// TIA Portal V15.1 export
// export: Created 2024-06-21T08:41:08.6869116Z, ExportSetting WithDefaults, DisplayName Totally Integrated Automation Portal, DisplayVersion V15.1 Update 5, DisplayName TIA Portal Openness, DisplayVersion V15.1 Update 5, DisplayName SINAMICS Startdrive Advanced, DisplayVersion V15.1, DisplayName G130, G150, S120, S150, SINAMICS MV, S210, DisplayVersion V15.1, DisplayName G110M, G120, G120C, G120D, G120P, DisplayVersion V15.1, DisplayName STEP 7 Professional, DisplayVersion V15.1 Update 5, DisplayName STEP 7 Safety, DisplayVersion V15.1, DisplayName WinCC Professional, DisplayVersion V15.1 Update 5, DisplayName SIMATIC Visualization Architect, DisplayVersion V15.1
FUNCTION "LGBHoist5PosIAnim" : Void   // FC6622, FBD
TITLE = LIAnimDWord / LGBHoist5PosIAnim
{ S7_Optimized_Access := 'TRUE' }
AUTHOR : VCC
FAMILY : Anim
NAME : SIAnim
VERSION : 0.1
// =============================================================================
// Handles the conversion from bits to one Word for simple icon Animation. 
// =============================================================================
// stored: AutoNumber false, IsIECCheckEnabled false, SetENOAutomatically False, UDAEnableTagReadback false
   VAR_INPUT
      I_OnPos : Bool;   // Set position / Set Position / On Position
      I_Active : Bool;   // Active
      I_Visible : Bool;   // ObjectVisible
      I_OutOfUse : Bool;   // Object out of use
      I_IntlkPos1 : Bool;   // Interlock for Set direction / Interlock for Position 1
      I_IntlkPos2 : Bool;   // Interlock for Set direction / Interlock for Position 2
      I_IntlkPos3 : Bool;   // Interlock for Reset direction / Interlock for Position 3
      I_IntlkPos4 : Bool;   // Interlock for Reset direction / Interlock for Position 4
      I_IntlkPos5 : Bool;   // Interlock for Reset direction / Interlock for Position 5
      I_IntlkPosMaint : Bool;   // Interlock for Reset direction / Interlock for Position Maintenance
      I_IntlkJog : Bool;   // Interlock for Reset direction / Interlock for Jog mode
      I_IntlkReferencing : Bool;   // Interlock for Reset direction / Interlock for Referencing mode
      I_VisibleIntlkPos1 : Bool;   // Interlock alarm for Set direction / Interlock Alarm for Set direction / Visible Interlock Position 1
      I_VisibleIntlkPos2 : Bool;   // Interlock alarm for Set direction / Interlock Alarm for Set direction / Visible Interlock Position 2
      I_VisibleIntlkPos3 : Bool;   // Interlock alarm for Reset direction / Interlock Alarm for Reset direction / Visible Interlock Position 3
      I_VisibleIntlkPos4 : Bool;   // Interlock alarm for Reset direction / Interlock Alarm for Reset direction / Visible Interlock Position 4
      I_VisibleIntlkPos5 : Bool;   // Interlock alarm for Reset direction / Interlock Alarm for Reset direction / Visible Interlock Position 5
      I_VisibleIntlkPosMaint : Bool;   // Interlock alarm for Reset direction / Interlock Alarm for Reset direction / Visible Interlock Position Maint
      I_ManualMode : Bool;   // Manual mode / Manual Mode
      I_FncSelInHMI : Bool;   // Manual selection from HMI
      I_AlarmA : Bool;   // AlarmA
      I_AlarmB : Bool;   // AlarmB
      I_AlarmC : Bool;   // AlarmC
      I_AlarmD : Bool;   // AlarmD
      I_SafetyOk : Bool;   // Safety Ok / Safety OK
      I_MotionStopNOk : Bool;   // Safety Ok / Motion Stop OK
   END_VAR
   VAR_OUTPUT
      H_IAnim : DWord;   // Icon animation Word / Icon Animation
   END_VAR
BEGIN

REGION Network 1: Icon animation Word / **** 1 - Inputs **** Set position / **** 1 - Inputs **** On position
   // Set Position / On position
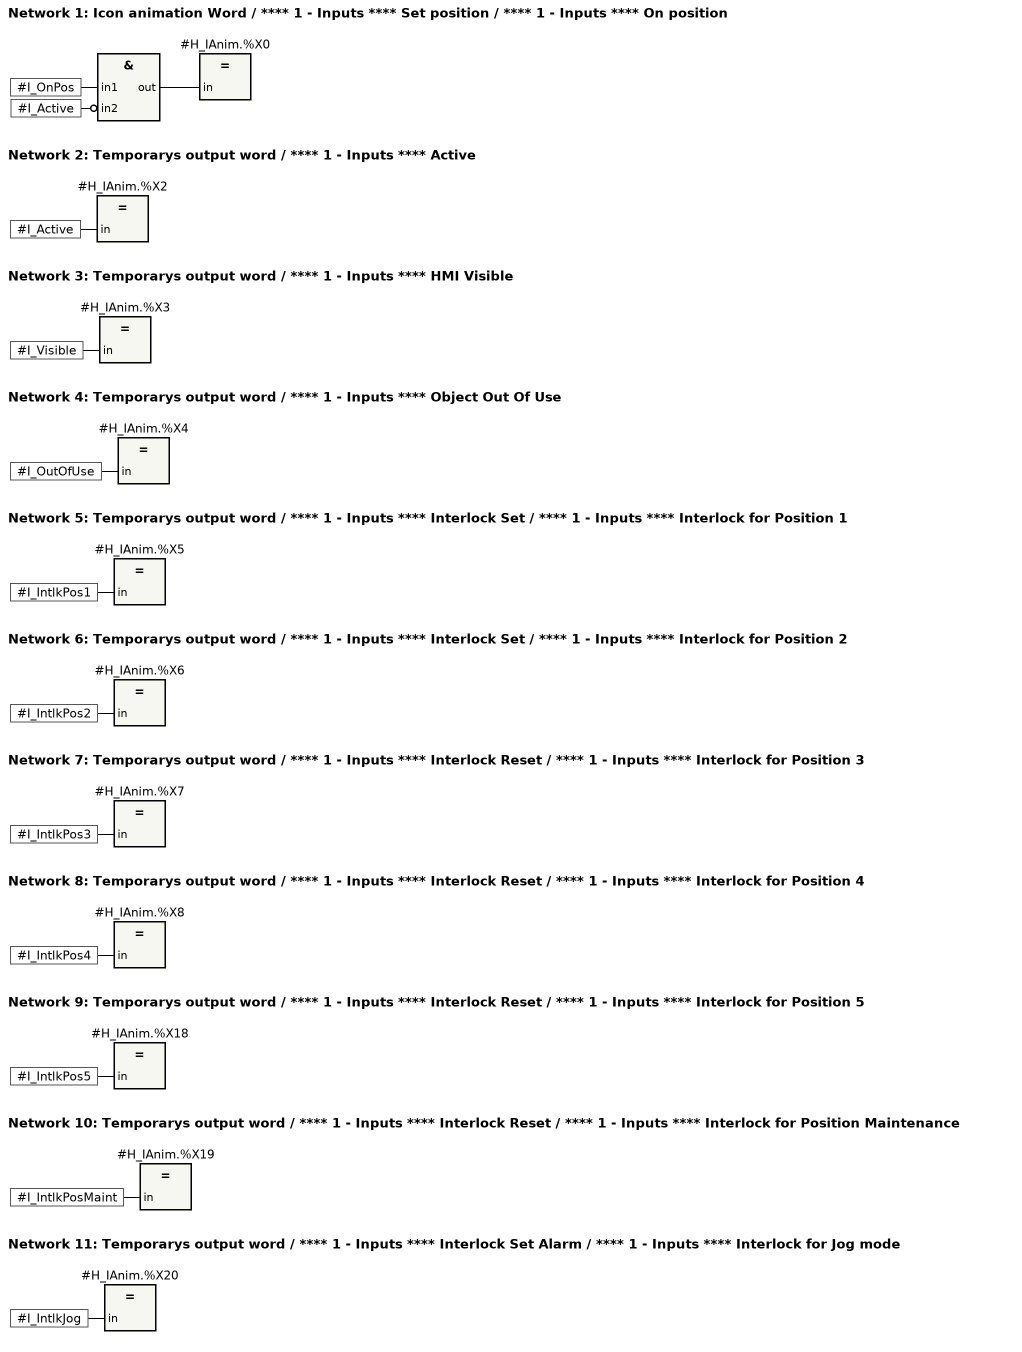
   #H_IAnim.%X0 := #I_OnPos AND NOT #I_Active;
END_REGION

REGION Network 2: Temporarys output word / **** 1 - Inputs **** Active
   // Active
   #H_IAnim.%X2 := #I_Active;
END_REGION

REGION Network 3: Temporarys output word / **** 1 - Inputs **** HMI Visible
   // HMI Visible
   #H_IAnim.%X3 := #I_Visible;
END_REGION

REGION Network 4: Temporarys output word / **** 1 - Inputs **** Object Out Of Use
   // Object out of use
   #H_IAnim.%X4 := #I_OutOfUse;
END_REGION

REGION Network 5: Temporarys output word / **** 1 - Inputs **** Interlock Set / **** 1 - Inputs **** Interlock for Position 1
   // Interlock Set / Interlock for Position 1
   #H_IAnim.%X5 := #I_IntlkPos1;
END_REGION

REGION Network 6: Temporarys output word / **** 1 - Inputs **** Interlock Set / **** 1 - Inputs **** Interlock for Position 2
   // Interlock Set / Interlock for Position 2
   #H_IAnim.%X6 := #I_IntlkPos2;
END_REGION

REGION Network 7: Temporarys output word / **** 1 - Inputs **** Interlock Reset / **** 1 - Inputs **** Interlock for Position 3
   // Interlock Reset / Interlock for Position 3
   #H_IAnim.%X7 := #I_IntlkPos3;
END_REGION

REGION Network 8: Temporarys output word / **** 1 - Inputs **** Interlock Reset / **** 1 - Inputs **** Interlock for Position 4
   // Interlock Reset / Interlock for Position 4
   #H_IAnim.%X8 := #I_IntlkPos4;
END_REGION

REGION Network 9: Temporarys output word / **** 1 - Inputs **** Interlock Reset / **** 1 - Inputs **** Interlock for Position 5
   // Interlock Reset / Interlock for Position 5
   #H_IAnim.%X18 := #I_IntlkPos5;
END_REGION

REGION Network 10: Temporarys output word / **** 1 - Inputs **** Interlock Reset / **** 1 - Inputs **** Interlock for Position Maintenance
   // Interlock Reset / Interlock for Position Maintenance
   #H_IAnim.%X19 := #I_IntlkPosMaint;
END_REGION

REGION Network 11: Temporarys output word / **** 1 - Inputs **** Interlock Set Alarm / **** 1 - Inputs **** Interlock for Jog mode
   // Interlock Set Alarm / Interlock for Jog mode
   #H_IAnim.%X20 := #I_IntlkJog;
END_REGION

REGION Network 12: Temporarys output word / **** 1 - Inputs **** Interlock Set Alarm / **** 1 - Inputs **** Interlock for Referencing mode
   // Interlock Set Alarm / Interlock for Referencing mode
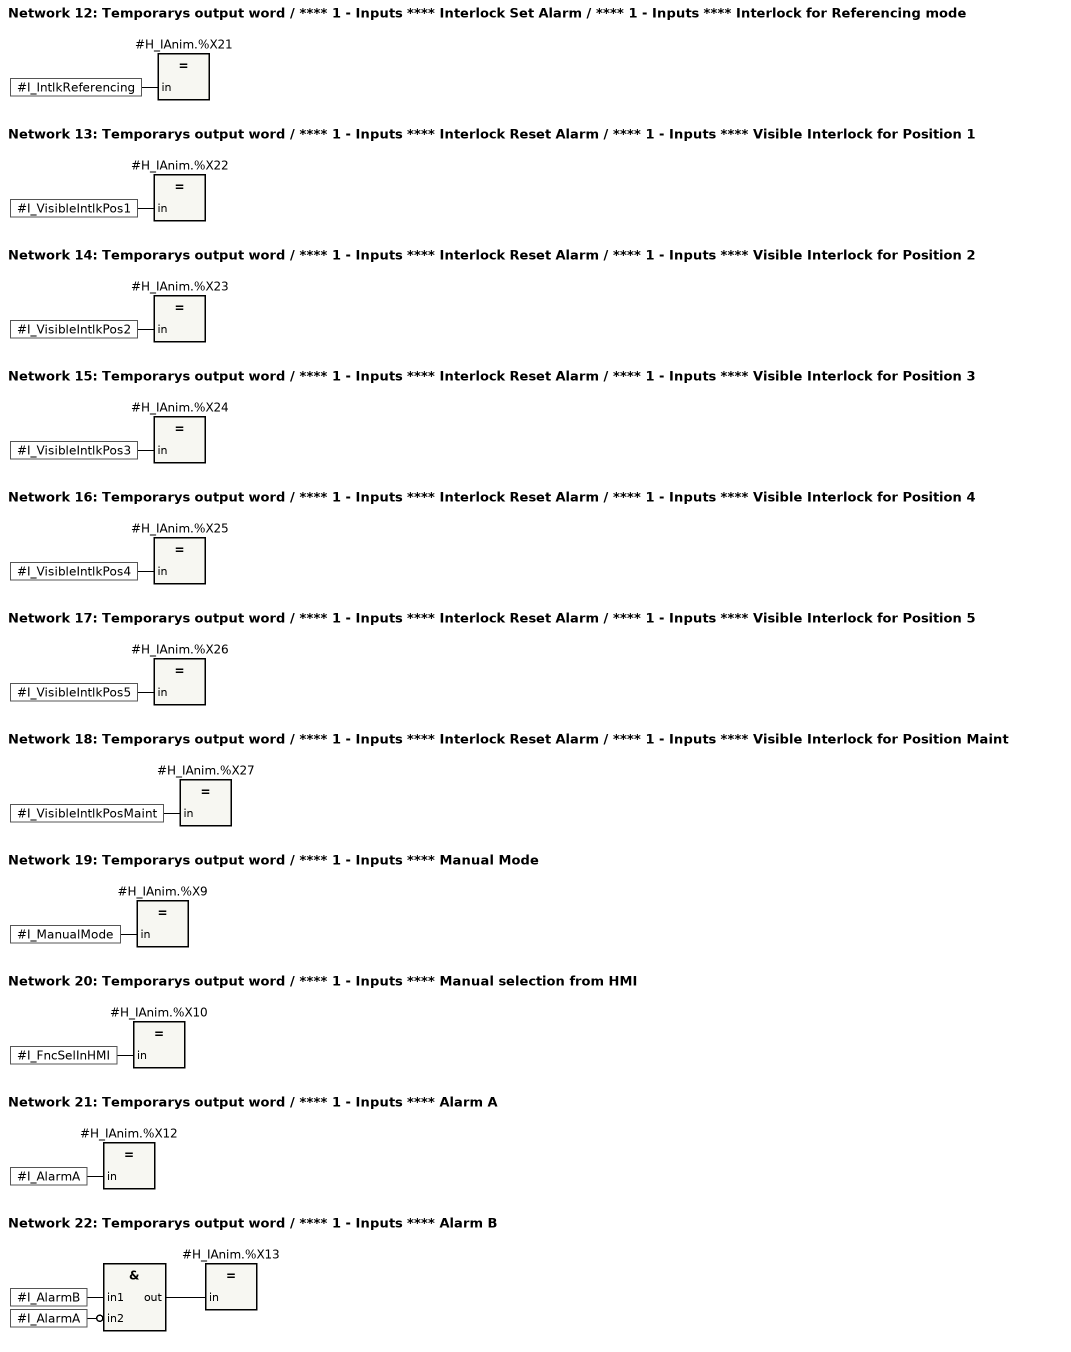
   #H_IAnim.%X21 := #I_IntlkReferencing;
END_REGION

REGION Network 13: Temporarys output word / **** 1 - Inputs **** Interlock Reset Alarm / **** 1 - Inputs **** Visible Interlock for Position 1
   // Interlock Reset Alarm / Visible Interlock for Position 1
   #H_IAnim.%X22 := #I_VisibleIntlkPos1;
END_REGION

REGION Network 14: Temporarys output word / **** 1 - Inputs **** Interlock Reset Alarm / **** 1 - Inputs **** Visible Interlock for Position 2
   // Interlock Reset Alarm / Visible Interlock for Position 2
   #H_IAnim.%X23 := #I_VisibleIntlkPos2;
END_REGION

REGION Network 15: Temporarys output word / **** 1 - Inputs **** Interlock Reset Alarm / **** 1 - Inputs **** Visible Interlock for Position 3
   // Interlock Reset Alarm / Visible Interlock for Position 3
   #H_IAnim.%X24 := #I_VisibleIntlkPos3;
END_REGION

REGION Network 16: Temporarys output word / **** 1 - Inputs **** Interlock Reset Alarm / **** 1 - Inputs **** Visible Interlock for Position 4
   // Interlock Reset Alarm / Visible Interlock for Position 4
   #H_IAnim.%X25 := #I_VisibleIntlkPos4;
END_REGION

REGION Network 17: Temporarys output word / **** 1 - Inputs **** Interlock Reset Alarm / **** 1 - Inputs **** Visible Interlock for Position 5
   // Interlock Reset Alarm / Visible Interlock for Position 5
   #H_IAnim.%X26 := #I_VisibleIntlkPos5;
END_REGION

REGION Network 18: Temporarys output word / **** 1 - Inputs **** Interlock Reset Alarm / **** 1 - Inputs **** Visible Interlock for Position Maint
   // Interlock Reset Alarm / Visible Interlock for Position Maintenance
   #H_IAnim.%X27 := #I_VisibleIntlkPosMaint;
END_REGION

REGION Network 19: Temporarys output word / **** 1 - Inputs **** Manual Mode
   // Manual Mode
   #H_IAnim.%X9 := #I_ManualMode;
END_REGION

REGION Network 20: Temporarys output word / **** 1 - Inputs **** Manual selection from HMI
   // Manual selection from HMI
   #H_IAnim.%X10 := #I_FncSelInHMI;
END_REGION

REGION Network 21: Temporarys output word / **** 1 - Inputs **** Alarm A
   // Alarm A
   #H_IAnim.%X12 := #I_AlarmA;
END_REGION

REGION Network 22: Temporarys output word / **** 1 - Inputs **** Alarm B
   // Alarm B
   #H_IAnim.%X13 := #I_AlarmB AND NOT #I_AlarmA;
END_REGION

REGION Network 23: Temporarys output word / **** 1 - Inputs **** Alarm C
   // Alarm C
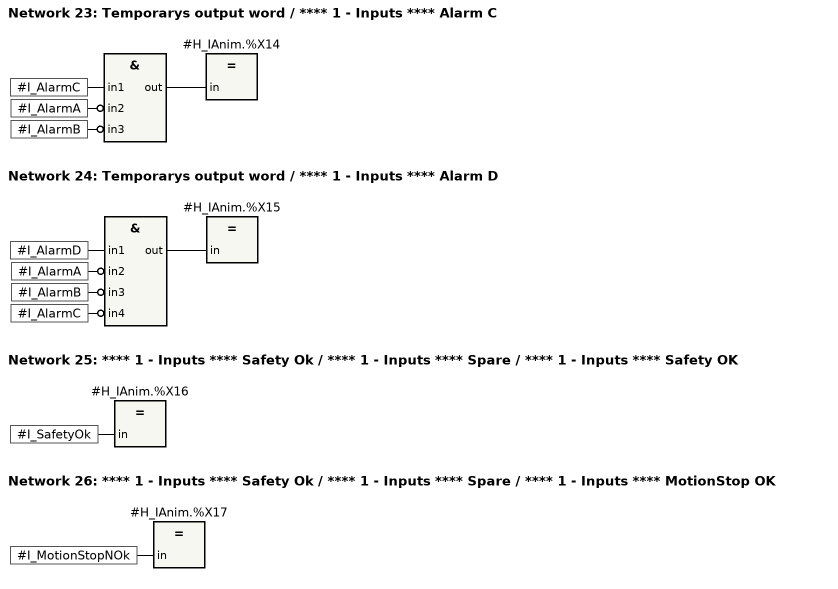
   #H_IAnim.%X14 := #I_AlarmC AND NOT #I_AlarmA AND NOT #I_AlarmB;
END_REGION

REGION Network 24: Temporarys output word / **** 1 - Inputs **** Alarm D
   // Alarm D
   #H_IAnim.%X15 := #I_AlarmD AND NOT #I_AlarmA AND NOT #I_AlarmB AND NOT #I_AlarmC;
END_REGION

REGION Network 25: **** 1 - Inputs **** Safety Ok / **** 1 - Inputs **** Spare / **** 1 - Inputs **** Safety OK
   // Safety Ok / Spare / Safety OK
   #H_IAnim.%X16 := #I_SafetyOk;
END_REGION

REGION Network 26: **** 1 - Inputs **** Safety Ok / **** 1 - Inputs **** Spare / **** 1 - Inputs **** MotionStop OK
   // Safety Ok / Spare / MotionStop OK
   #H_IAnim.%X17 := #I_MotionStopNOk;
END_REGION
END_FUNCTION
